FUNCTION F_TIME_ARG : ST_Arg
VAR_INPUT
	tInput : TIME;
END_VAR
VAR
	stArg : ST_Arg;
	sysVar_Info : __SYSTEM.VAR_INFO;
END_VAR

sysVar_Info 	:= __VARINFO(tInput);
stArg.TypeClass := sysVar_Info.TypeClass;
stArg.pValue 	:= 0;
stArg.diSize 	:= SIZEOF(tInput);
stArg.sValue 	:= TO_STRING(tInput); 
F_TIME_ARG := stArg;

END_FUNCTION

(* stored: Version 1.1.0.1, ProductVersion 3.1.4024.4
   POU F_TIME_ARG: Id {6ba44874-19c9-499f-9799-3a32352fd2b9}, SpecialFunc None *)
